{attribute 'qualified_only'}
{attribute 'strict'}
TYPE E_ComauMode :
(
	SETTLED := 0,
	REMOTE,
	MOTION_COMP
) DINT;
END_TYPE

(* stored: Version 1.1.0.1, ProductVersion 3.1.4022.18
   DUT E_ComauMode: Id {22f08a95-8072-4f02-bacf-d56adc38aaa2} *)
